// TIA Portal V16 export
// export: Created 2022-11-14T17:35:39.342922Z, ExportSetting WithDefaults, DisplayName Totally Integrated Automation Portal, DisplayVersion V16, DisplayName TIA Portal Version Control Interface, DisplayVersion V16, DisplayName TIA Portal Openness, DisplayVersion V16, DisplayName STEP 7 Professional, DisplayVersion V16, DisplayName STEP 7 Safety, DisplayVersion V16, DisplayName WinCC Advanced, DisplayVersion V16
DATA_BLOCK "Timer"   // DB2
{ S7_Optimized_Access := 'TRUE' }
VERSION : 0.0
// stored: AutoNumber false, IsOnlyStoredInLoadMemory false, IsRetainMemResEnabled false, IsWriteProtectedInAS false, MemoryReserve 100
   VAR
      T0 { S7_SetPoint := 'True'} : IEC_TIMER;   // Delay on pallet positioning
      T1 { S7_SetPoint := 'True'} : IEC_TIMER;   // Timer for acoustic siren
      T2 { S7_SetPoint := 'True'} : IEC_TIMER;   // Timer for restart after emergency
      T3 { S7_SetPoint := 'True'} : IEC_TIMER;   // Timer to reset emergency
      T4 { S7_SetPoint := 'True'} : IEC_TIMER;   // Timer to reset the cycles
      T5 { S7_SetPoint := 'True'} : IEC_TIMER;   // Delay for backward on table rotation inverter
      T6 { S7_SetPoint := 'True'} : IEC_TIMER;   // Delay for forward on table rotation inverter
      T7 { S7_SetPoint := 'True'} : IEC_TIMER;   // Timeout for table phase
      T8 { S7_SetPoint := 'True'} : IEC_TIMER;   // Table rotation speed timer
      T9 { S7_SetPoint := 'True'} : IEC_TIMER;   // Timer SA type for spool carriage motor
      T10 { S7_SetPoint := 'True'} : IEC_TIMER;   // Timer SA type for table rotation motor
      T11 { S7_SetPoint := 'True'} : IEC_TIMER;   // Timer SA type for spool carriage downward
      T12 { S7_SetPoint := 'True'} : IEC_TIMER;   // Timer SA type for spool carriage upward
      T13 { S7_SetPoint := 'True'} : IEC_TIMER;   // Timer SA type for top carriage motor
      T14 { S7_SetPoint := 'True'} : IEC_TIMER;   // Delay for forward on spool carriage and machine conveyor inverter
      T15 { S7_SetPoint := 'True'} : IEC_TIMER;   // Timer for lifter upward
      T16 { S7_SetPoint := 'True'} : IEC_TIMER;   // Timeout for pallet lifter upward/downward
      T17 { S7_SetPoint := 'True'} : IEC_TIMER;   // Time for pressure plate downward
      T18 { S7_SetPoint := 'True'} : IEC_TIMER;   // Timeout for pressure plate upward/downward
      T19 { S7_SetPoint := 'True'} : IEC_TIMER;   // Delay for backward on spool carriage and machine conveyor inverter
      T20 { S7_SetPoint := 'True'} : IEC_TIMER;   // Delay for table rotation deceleration
      T21 { S7_SetPoint := 'True'} : IEC_TIMER;   // Film broken delay for spool carriage
      T22 { S7_SetPoint := 'True'} : IEC_TIMER;   // Delay for pressure plate positioning on pallet
      T23 { S7_SetPoint := 'True'} : IEC_TIMER;   // Timer SA type for conveyor motor
      T24 { S7_SetPoint := 'True'} : IEC_TIMER;   // Delay on pallet positioning left
      T25 { S7_SetPoint := 'True'} : IEC_TIMER;   // Delay on machine conveyor stop
      T26 { S7_SetPoint := 'True'} : IEC_TIMER;   // Delay to load/unload pallet simultaneously
      T27 { S7_SetPoint := 'True'} : IEC_TIMER;   // Delay to have outfeed control free
      T28 { S7_SetPoint := 'True'} : IEC_TIMER;   // Timer for end of transfer signal
      T29 { S7_SetPoint := 'True'} : IEC_TIMER;   // Timer to check spool carriage encoder
      T30 { S7_SetPoint := 'True'} : IEC_TIMER;   // Timer to check spool carriage encoder
      T31 { S7_SetPoint := 'True'} : IEC_TIMER;   // Time to record spool carriage movement speed
      T32 { S7_SetPoint := 'True'} : IEC_TIMER;   // Timeout for single or lower(double) rope unit open/close
      T33 { S7_SetPoint := 'True'} : IEC_TIMER;   // Timer for outfeed rotating table control engaged
      T34 { S7_SetPoint := 'True'} : IEC_TIMER;   // Timer for prestretch restart
      T35 { S7_SetPoint := 'True'} : IEC_TIMER;   // Delay to open single or lower(double) rope unit
      T36 { S7_SetPoint := 'True'} : IEC_TIMER;   // Timeout for welder unit upward/downward
      T37 { S7_SetPoint := 'True'} : IEC_TIMER;   // Timeout for welder contrast downward
      T38 { S7_SetPoint := 'True'} : IEC_TIMER;   // Timeout for welder contrast upward
      T39 { S7_SetPoint := 'True'} : IEC_TIMER;   // Timeout for clamp upward/downward
      T40 { S7_SetPoint := 'True'} : IEC_TIMER;   // Timeout for clamp open/close
      T41 { S7_SetPoint := 'True'} : IEC_TIMER;   // Welding timer for welder
      T42 { S7_SetPoint := 'True'} : IEC_TIMER;   // Cutting timer
      T43 { S7_SetPoint := 'True'} : IEC_TIMER;   // Welder cooler timer
      T44 { S7_SetPoint := 'True'} : IEC_TIMER;   // Timer to check welder circuit 1 (current on)
      T45 { S7_SetPoint := 'True'} : IEC_TIMER;   // Timer to check welder circuit 2 (current off)
      T46 { S7_SetPoint := 'True'} : IEC_TIMER;   // Spring clamp up
      T47 { S7_SetPoint := 'True'} : IEC_TIMER;   // Welder contrast up
      T48 { S7_SetPoint := 'True'} : IEC_TIMER;   // Spring clamp open
      T49 { S7_SetPoint := 'True'} : IEC_TIMER;   // Welder and cut unit up
      T50 { S7_SetPoint := 'True'} : IEC_TIMER;   // Timer for encoder check
      T51 { S7_SetPoint := 'True'} : IEC_TIMER;   // Timer for display comunication control
      T52 { S7_SetPoint := 'True'} : IEC_TIMER;   // Timer to return to page 1 after 3 minutes
      T53 { S7_SetPoint := 'True'} : IEC_TIMER;   // Delay for test cycle
      T54 { S7_SetPoint := 'True'} : IEC_TIMER;   // Timer to reset infeed safety barrier
      T55 { S7_SetPoint := 'True'} : IEC_TIMER;   // Timer to reset infeed safety barrier
      T56 { S7_SetPoint := 'True'} : IEC_TIMER;   // Timer to reset outfeed safety barrier
      T57 { S7_SetPoint := 'True'} : IEC_TIMER;   // Timer to reset outfeed safety barrier
      T58 { S7_SetPoint := 'True'} : IEC_TIMER;   // Delay for infeed safety barrier muting photocell
      T59 { S7_SetPoint := 'True'} : IEC_TIMER;   // Delay for outfeed safety barrier muting photocell
      T60 { S7_SetPoint := 'True'} : IEC_TIMER;   // Delay for spool carriage downward for film tail
      T61 { S7_SetPoint := 'True'} : IEC_TIMER;   // Delay to open clamp during wrapping cycle
      T62 { S7_SetPoint := 'True'} : IEC_TIMER;   // Timer for table rotation forward on twist
      T63 { S7_SetPoint := 'True'} : IEC_TIMER;   // Timer SA type for top carriage upward
      T64 { S7_SetPoint := 'True'} : IEC_TIMER;   // Timer SA type for top carriage downward
      T65 { S7_SetPoint := 'True'} : IEC_TIMER;   // Delay on safety for top carriage movement
      T66 { S7_SetPoint := 'True'} : IEC_TIMER;   // Timer to check top film presence
      T67 { S7_SetPoint := 'True'} : IEC_TIMER;   // Timer to check top film presence
      T68 { S7_SetPoint := 'True'} : IEC_TIMER;   // Timeout for top film cutter forward/backward
      T69 { S7_SetPoint := 'True'} : IEC_TIMER;   // Timeout for clamp to lift top film open/close
      T70 { S7_SetPoint := 'True'} : IEC_TIMER;   // Timeout for clamp to block top film open/close
      T71 { S7_SetPoint := 'True'} : IEC_TIMER;   // Timeout for top carriage forward/backward movement
      T72 { S7_SetPoint := 'True'} : IEC_TIMER;   // Timeout for top carriage forward/backward movement
      T73 { S7_SetPoint := 'True'} : IEC_TIMER;   // Timeout for top carriage upward/downward movement
      T74 { S7_SetPoint := 'True'} : IEC_TIMER;   // Timeout for top carriage upward/downward movement
      T75 { S7_SetPoint := 'True'} : IEC_TIMER;   // Delay for spool carriage downward during top cycle
      T76 { S7_SetPoint := 'True'} : IEC_TIMER;   // Claw clamp closed
      T77 { S7_SetPoint := 'True'} : IEC_TIMER;   // Timeout for welder and cut unit forward/backward
      T78 { S7_SetPoint := 'True'} : IEC_TIMER;   // Delay to open upper(double) rope unit
      T79 { S7_SetPoint := 'True'} : IEC_TIMER;   // Timer SA type for table rotation brake
      T80 { S7_SetPoint := 'True'} : IEC_TIMER;   // Timer for spool carriage movement speed
      T81 { S7_SetPoint := 'True'} : IEC_TIMER;   // Claw clamp closed
      T82 { S7_SetPoint := 'True'} : IEC_TIMER;   // Timeout for welder and cut unit forward/backward
      T83 { S7_SetPoint := 'True'} : IEC_TIMER;   // Delay between airblow and clamp
      T84 { S7_SetPoint := 'True'} : IEC_TIMER;   // Timer for table rotation speed
      T85 { S7_SetPoint := 'True'} : IEC_TIMER;   // Delay on infeed conveyor stop
      T86 { S7_SetPoint := 'True'} : IEC_TIMER;   // Delay for prestretch during acceleration
      T87 { S7_SetPoint := 'True'} : IEC_TIMER;   // Timer for slow conveyor manual movement
      T88 { S7_SetPoint := 'True'} : IEC_TIMER;
      T89 { S7_SetPoint := 'True'} : IEC_TIMER;   // Timer for wrong pallet positioning without outfeed control
      T90 { S7_SetPoint := 'True'} : IEC_TIMER;   // Timer for spool carriage upward for table cycle
      T91 { S7_SetPoint := 'True'} : IEC_TIMER;   // Delay to close clamp after cutter forward
      T92 { S7_SetPoint := 'True'} : IEC_TIMER;   // Delay for contrast downward
      T93 { S7_SetPoint := 'True'} : IEC_TIMER;
      T94 { S7_SetPoint := 'True'} : IEC_TIMER;
      T95 { S7_SetPoint := 'True'} : IEC_TIMER;
      T96 { S7_SetPoint := 'True'} : IEC_TIMER;   // Timeout for fire door pos.4-5 opening
      T97 { S7_SetPoint := 'True'} : IEC_TIMER;   // Delay conveyor manual movement
      T98 { S7_SetPoint := 'True'} : IEC_TIMER;   // Delay start cycle pos.1
      T99 { S7_SetPoint := 'True'} : IEC_TIMER;   // Time to load with forklift
      T100 { S7_SetPoint := 'True'} : IEC_TIMER;   // Timer for end of pallet transfer in infeed signal
      T101 { S7_SetPoint := 'True'} : IEC_TIMER;   // Timeout for conveyor pos 01
      T102 { S7_SetPoint := 'True'} : IEC_TIMER;   // Time to load with forklift
      T103 { S7_SetPoint := 'True'} : IEC_TIMER;   // Timeout for conveyor pos 02
      T104 { S7_SetPoint := 'True'} : IEC_TIMER;
      T105 { S7_SetPoint := 'True'} : IEC_TIMER;   // Timeout for conveyor pos 04
      T106 { S7_SetPoint := 'True'} : IEC_TIMER;   // Timeout for conveyor pos 03
      T107 { S7_SetPoint := 'True'} : IEC_TIMER;   // Time for pallet unload with forklift
      T108 { S7_SetPoint := 'True'} : IEC_TIMER;   // Delay Button Stop cycle support memory
      T109 { S7_SetPoint := 'True'} : IEC_TIMER;   // Time for pallet load with forklift from reverse
      T110 { S7_SetPoint := 'True'} : IEC_TIMER;   // Timer to reset machine and cycle
      T111 { S7_SetPoint := 'True'} : IEC_TIMER;   // Delay timer for lifter pos.2 low position
      T112 { S7_SetPoint := 'True'} : IEC_TIMER;   // Delay timer for lifter pos.2 up position
      T113 { S7_SetPoint := 'True'} : IEC_TIMER;   // Delay timer pallet positioned on lifter pos.2
      T114 { S7_SetPoint := 'True'} : IEC_TIMER;   // Timer SA for lifter in top position
      T115 { S7_SetPoint := 'True'} : IEC_TIMER;   // Timeout for conveyor pos.2
      T116 { S7_SetPoint := 'True'} : IEC_TIMER;   // Timeout for lifter pos.2 upstroke
      T117 { S7_SetPoint := 'True'} : IEC_TIMER;   // Timeout for lifter pos.2 downstroke
      T118 { S7_SetPoint := 'True'} : IEC_TIMER;   // Timer to filter lifter pos.2 in up position
      T119 { S7_SetPoint := 'True'} : IEC_TIMER;
      T120 { S7_SetPoint := 'True'} : IEC_TIMER;   // Timer to check conveyor encoder
      T121 { S7_SetPoint := 'True'} : IEC_TIMER;   // Timer to check conveyor encoder
      T122 { S7_SetPoint := 'True'} : IEC_TIMER;
      T123 { S7_SetPoint := 'True'} : IEC_TIMER;
      T124 { S7_SetPoint := 'True'} : IEC_TIMER;
      T125 { S7_SetPoint := 'True'} : IEC_TIMER;
      T126 { S7_SetPoint := 'True'} : IEC_TIMER;
      T127 { S7_SetPoint := 'True'} : IEC_TIMER;   // Delay to have outfeed rotating arm control free from reverse
      T128 { S7_SetPoint := 'True'} : IEC_TIMER;   // Timer for end of transfer signal from reverse
      T129 { S7_SetPoint := 'True'} : IEC_TIMER;
      T130 { S7_SetPoint := 'True'} : IEC_TIMER;
      T131 { S7_SetPoint := 'True'} : IEC_TIMER;
      T132 { S7_SetPoint := 'True'} : IEC_TIMER;   // Timeout for single or lower(double) rope unit open/close
      T133 { S7_SetPoint := 'True'} : IEC_TIMER;
      T134 { S7_SetPoint := 'True'} : IEC_TIMER;
      T135 { S7_SetPoint := 'True'} : IEC_TIMER;   // Delay to open single or lower(double) rope unit
      T136 { S7_SetPoint := 'True'} : IEC_TIMER;
      T137 { S7_SetPoint := 'True'} : IEC_TIMER;
      T138 { S7_SetPoint := 'True'} : IEC_TIMER;
      T139 { S7_SetPoint := 'True'} : IEC_TIMER;   // Delay for top carriage forward stop (Top)
      T140 { S7_SetPoint := 'True'} : IEC_TIMER;   // Delay for top carriage backward stop (Top)
      T141 { S7_SetPoint := 'True'} : IEC_TIMER;
      T142 { S7_SetPoint := 'True'} : IEC_TIMER;   // Delay for top carriage down to release top film (Top)
      T143 { S7_SetPoint := 'True'} : IEC_TIMER;   // Delay to release top film from clamp (Top)
      T144 { S7_SetPoint := 'True'} : IEC_TIMER;   // Timer 1 for top film broken (Top)
      T145 { S7_SetPoint := 'True'} : IEC_TIMER;   // Timer 2 for top film broken (Top)
      T146 { S7_SetPoint := 'True'} : IEC_TIMER;   // Delay to stop top carriage forward for top film broken (Top)
      T147 { S7_SetPoint := 'True'} : IEC_TIMER;   // Delay to stop top carriage against vibration (Top)
      T148 { S7_SetPoint := 'True'} : IEC_TIMER;   // Timeout for top cutter (Top)
      T149 { S7_SetPoint := 'True'} : IEC_TIMER;   // Timeout for clamp to pull top film (Top)
      T150 { S7_SetPoint := 'True'} : IEC_TIMER;   // Timeout for clamp to block top film (Top)
      T151 { S7_SetPoint := 'True'} : IEC_TIMER;   // Timer SA type for top brake (Top)
      T152 { S7_SetPoint := 'True'} : IEC_TIMER;   // Timer for top brake control (Top)
      T153 { S7_SetPoint := 'True'} : IEC_TIMER;
      T154 { S7_SetPoint := 'True'} : IEC_TIMER;
      T155 { S7_SetPoint := 'True'} : IEC_TIMER;   // Timeout for conveyor pos 03
      T156 { S7_SetPoint := 'True'} : IEC_TIMER;   // Timeout for conveyor pos 04
      T157 { S7_SetPoint := 'True'} : IEC_TIMER;   // Timeout for conveyor pos 05
      T158 { S7_SetPoint := 'True'} : IEC_TIMER;   // Timeout for conveyor pos 06
      T159 { S7_SetPoint := 'True'} : IEC_TIMER;   // Timeout for conveyor pos 07
      T160 { S7_SetPoint := 'True'} : IEC_TIMER;   // Timeout for conveyor pos 08
      T161 { S7_SetPoint := 'True'} : IEC_TIMER;
      T162 { S7_SetPoint := 'True'} : IEC_TIMER;
      T163 { S7_SetPoint := 'True'} : IEC_TIMER;   // Watchdog timer for network communication
      T164 { S7_SetPoint := 'True'} : IEC_TIMER;
      T165 { S7_SetPoint := 'True'} : IEC_TIMER;
      T166 { S7_SetPoint := 'True'} : IEC_TIMER;
      T167 { S7_SetPoint := 'True'} : IEC_TIMER;
      T168 { S7_SetPoint := 'True'} : IEC_TIMER;
      T169 { S7_SetPoint := 'True'} : IEC_TIMER;
      T170 { S7_SetPoint := 'True'} : IEC_TIMER;
      T171 { S7_SetPoint := 'True'} : IEC_TIMER;
      T172 { S7_SetPoint := 'True'} : IEC_TIMER;
      T173 { S7_SetPoint := 'True'} : IEC_TIMER;
      T174 { S7_SetPoint := 'True'} : IEC_TIMER;
      T175 { S7_SetPoint := 'True'} : IEC_TIMER;
      T176 { S7_SetPoint := 'True'} : IEC_TIMER;
      T177 { S7_SetPoint := 'True'} : IEC_TIMER;
      T178 { S7_SetPoint := 'True'} : IEC_TIMER;
      T179 { S7_SetPoint := 'True'} : IEC_TIMER;   // Delay for top pallet height reading photocell (fast cycle)
      T180 { S7_SetPoint := 'True'} : IEC_TIMER;
      T181 { S7_SetPoint := 'True'} : IEC_TIMER;
      T182 { S7_SetPoint := 'True'} : IEC_TIMER;
      T183 { S7_SetPoint := 'True'} : IEC_TIMER;
      T184 { S7_SetPoint := 'True'} : IEC_TIMER;
      T185 { S7_SetPoint := 'True'} : IEC_TIMER;
      T186 { S7_SetPoint := 'True'} : IEC_TIMER;
      T187 { S7_SetPoint := 'True'} : IEC_TIMER;
      T188 { S7_SetPoint := 'True'} : IEC_TIMER;
      T189 { S7_SetPoint := 'True'} : IEC_TIMER;
      T190 { S7_SetPoint := 'True'} : IEC_TIMER;
      T191 { S7_SetPoint := 'True'} : IEC_TIMER;
      T192 { S7_SetPoint := 'True'} : IEC_TIMER;
      T193 { S7_SetPoint := 'True'} : IEC_TIMER;
      T194 { S7_SetPoint := 'True'} : IEC_TIMER;
      T195 { S7_SetPoint := 'True'} : IEC_TIMER;
      T196 { S7_SetPoint := 'True'} : IEC_TIMER;
      T197 { S7_SetPoint := 'True'} : IEC_TIMER;
      T198 { S7_SetPoint := 'True'} : IEC_TIMER;
      T199 { S7_SetPoint := 'True'} : IEC_TIMER;
      T200 { S7_SetPoint := 'True'} : IEC_TIMER;   // T_InverterAlarm - Time to filter inverter alarms
      T201 { S7_SetPoint := 'True'} : IEC_TIMER;   // T_ProfinetDiag - Time to filter 'DeviceStates' diagnostic output (Profinet)
      T202 { S7_SetPoint := 'True'} : IEC_TIMER;   // Timer for U201 start command (after enable)
      T203 { S7_SetPoint := 'True'} : IEC_TIMER;   // Timer table backward
      T204 { S7_SetPoint := 'True'} : IEC_TIMER;   // Timer ciclo fiera
      T205 { S7_SetPoint := 'True'} : IEC_TIMER;   // TON per OFF1 U201
      T206 { S7_SetPoint := 'True'} : IEC_TIMER;   // TOF per OFF1 U201
      T207 { S7_SetPoint := 'True'} : IEC_TIMER;   // Timer coppia tavola
      T208 { S7_SetPoint := 'True'} : IEC_TIMER;   // T_ModbusErrors
      T209 { S7_SetPoint := 'True'} : IEC_TIMER;
      T210 { S7_SetPoint := 'True'} : IEC_TIMER;   // Time to filter contrast back sensor
      T211 { S7_SetPoint := 'True'} : IEC_TIMER;   // Timeout for welder contrast forward
      T212 { S7_SetPoint := 'True'} : IEC_TIMER;   // Timeout for welder contrast backward
      T213 { S7_SetPoint := 'True'} : IEC_TIMER;   // Timeout for (double) full rope unit open/close
      T214 { S7_SetPoint := 'True'} : IEC_TIMER;   // Delay to open single or lower(double) rope unit
      T215 { S7_SetPoint := 'True'} : IEC_TIMER;   // Time Contrast Backward
      T216 { S7_SetPoint := 'True'} : IEC_TIMER;   // Time Contrast Manual forward
   END_VAR
BEGIN
   T0.PT := T#0MS;
   T0.IN := FALSE;
   T1.PT := T#1S_200MS;
   T1.IN := FALSE;
   T2.PT := T#6S;
   T2.IN := TRUE;
   T3.PT := T#700MS;
   T3.IN := FALSE;
   T4.PT := T#2S;
   T4.IN := FALSE;
   T5.PT := T#800MS;
   T5.IN := FALSE;
   T6.PT := T#800MS;
   T6.IN := FALSE;
   T7.PT := T#50S;
   T7.IN := FALSE;
   T8.PT := T#1M_39S;
   T8.IN := FALSE;
   T9.PT := T#700MS;
   T9.IN := FALSE;
   T10.PT := T#2S;
   T10.IN := FALSE;
   T11.PT := T#500MS;
   T11.IN := FALSE;
   T12.PT := T#500MS;
   T12.IN := FALSE;
   T13.PT := T#0MS;
   T13.IN := FALSE;
   T14.PT := T#200MS;
   T14.IN := FALSE;
   T15.PT := T#0MS;
   T15.IN := FALSE;
   T16.PT := T#0MS;
   T16.IN := FALSE;
   T17.PT := T#0MS;
   T17.IN := FALSE;
   T18.PT := T#0MS;
   T18.IN := FALSE;
   T19.PT := T#200MS;
   T19.IN := FALSE;
   T20.PT := T#0MS;
   T20.IN := FALSE;
   T21.PT := T#2S;
   T21.IN := FALSE;
   T22.PT := T#0MS;
   T22.IN := FALSE;
   T23.PT := T#0MS;
   T23.IN := FALSE;
   T24.PT := T#0MS;
   T24.IN := FALSE;
   T25.PT := T#0MS;
   T25.IN := FALSE;
   T26.PT := T#0MS;
   T26.IN := FALSE;
   T27.PT := T#1S_500MS;
   T27.IN := TRUE;
   T28.PT := T#2S;
   T28.IN := TRUE;
   T29.PT := T#0MS;
   T29.IN := FALSE;
   T30.PT := T#3S;
   T30.IN := FALSE;
   T31.PT := T#0MS;
   T31.IN := FALSE;
   T32.PT := T#0MS;
   T32.IN := FALSE;
   T33.PT := T#0MS;
   T33.IN := FALSE;
   T34.PT := T#0MS;
   T34.IN := FALSE;
   T35.PT := T#0MS;
   T35.IN := FALSE;
   T36.PT := T#0MS;
   T36.IN := FALSE;
   T37.PT := T#0MS;
   T37.IN := FALSE;
   T38.PT := T#10S;
   T38.IN := FALSE;
   T39.PT := T#0MS;
   T39.IN := FALSE;
   T40.PT := T#0MS;
   T40.IN := FALSE;
   T41.PT := T#650MS;
   T41.IN := FALSE;
   T42.PT := T#3S;
   T42.IN := FALSE;
   T43.PT := T#0MS;
   T43.IN := FALSE;
   T44.PT := T#3S_500MS;
   T44.IN := FALSE;
   T45.PT := T#1S;
   T45.IN := FALSE;
   T46.PT := T#0MS;
   T46.IN := FALSE;
   T47.PT := T#500MS;
   T47.IN := TRUE;
   T48.PT := T#0MS;
   T48.IN := FALSE;
   T49.PT := T#0MS;
   T49.IN := FALSE;
   T50.PT := T#0MS;
   T50.IN := FALSE;
   T51.PT := T#4S;
   T51.IN := TRUE;
   T52.PT := T#0MS;
   T52.IN := FALSE;
   T53.PT := T#0MS;
   T53.IN := TRUE;
   T54.PT := T#0MS;
   T54.IN := FALSE;
   T55.PT := T#0MS;
   T55.IN := FALSE;
   T56.PT := T#0MS;
   T56.IN := FALSE;
   T57.PT := T#0MS;
   T57.IN := FALSE;
   T58.PT := T#0MS;
   T58.IN := FALSE;
   T59.PT := T#0MS;
   T59.IN := FALSE;
   T60.PT := T#0MS;
   T60.IN := FALSE;
   T61.PT := T#0MS;
   T61.IN := FALSE;
   T62.PT := T#0MS;
   T62.IN := FALSE;
   T63.PT := T#0MS;
   T63.IN := FALSE;
   T64.PT := T#0MS;
   T64.IN := FALSE;
   T65.PT := T#0MS;
   T65.IN := FALSE;
   T66.PT := T#0MS;
   T66.IN := FALSE;
   T67.PT := T#0MS;
   T67.IN := FALSE;
   T68.PT := T#0MS;
   T68.IN := FALSE;
   T69.PT := T#0MS;
   T69.IN := FALSE;
   T70.PT := T#0MS;
   T70.IN := FALSE;
   T71.PT := T#0MS;
   T71.IN := FALSE;
   T72.PT := T#0MS;
   T72.IN := FALSE;
   T73.PT := T#0MS;
   T73.IN := FALSE;
   T74.PT := T#0MS;
   T74.IN := FALSE;
   T75.PT := T#0MS;
   T75.IN := FALSE;
   T76.PT := T#0MS;
   T76.IN := FALSE;
   T77.PT := T#0MS;
   T77.IN := FALSE;
   T78.PT := T#0MS;
   T78.IN := FALSE;
   T79.PT := T#2S;
   T79.IN := FALSE;
   T80.PT := T#1S;
   T80.IN := TRUE;
   T81.PT := T#700MS;
   T81.IN := TRUE;
   T82.PT := T#10S;
   T82.IN := FALSE;
   T83.PT := T#500MS;
   T83.IN := FALSE;
   T84.PT := T#400MS;
   T84.IN := TRUE;
   T85.PT := T#0MS;
   T85.IN := FALSE;
   T86.PT := T#300MS;
   T86.IN := FALSE;
   T87.PT := T#0MS;
   T87.IN := FALSE;
   T88.PT := T#0MS;
   T88.IN := FALSE;
   T89.PT := T#0MS;
   T89.IN := FALSE;
   T90.PT := T#2S;
   T90.IN := FALSE;
   T91.PT := T#1S;
   T91.IN := FALSE;
   T92.PT := T#0MS;
   T92.IN := FALSE;
   T93.PT := T#0MS;
   T93.IN := FALSE;
   T94.PT := T#0MS;
   T94.IN := FALSE;
   T95.PT := T#0MS;
   T95.IN := FALSE;
   T96.PT := T#0MS;
   T96.IN := FALSE;
   T97.PT := T#0MS;
   T97.IN := FALSE;
   T98.PT := T#0MS;
   T98.IN := FALSE;
   T99.PT := T#0MS;
   T99.IN := FALSE;
   T100.PT := T#0MS;
   T100.IN := FALSE;
   T101.PT := T#0MS;
   T101.IN := FALSE;
   T102.PT := T#0MS;
   T102.IN := FALSE;
   T103.PT := T#0MS;
   T103.IN := FALSE;
   T104.PT := T#0MS;
   T104.IN := FALSE;
   T105.PT := T#0MS;
   T105.IN := FALSE;
   T106.PT := T#0MS;
   T106.IN := FALSE;
   T107.PT := T#0MS;
   T107.IN := FALSE;
   T108.PT := T#0MS;
   T108.IN := FALSE;
   T109.PT := T#0MS;
   T109.IN := FALSE;
   T110.PT := T#0MS;
   T110.IN := FALSE;
   T111.PT := T#0MS;
   T111.IN := FALSE;
   T112.PT := T#0MS;
   T112.IN := FALSE;
   T113.PT := T#0MS;
   T113.IN := FALSE;
   T114.PT := T#0MS;
   T114.IN := FALSE;
   T115.PT := T#0MS;
   T115.IN := FALSE;
   T116.PT := T#0MS;
   T116.IN := FALSE;
   T117.PT := T#0MS;
   T117.IN := FALSE;
   T118.PT := T#0MS;
   T118.IN := FALSE;
   T119.PT := T#0MS;
   T119.IN := FALSE;
   T120.PT := T#0MS;
   T120.IN := FALSE;
   T121.PT := T#0MS;
   T121.IN := FALSE;
   T122.PT := T#0MS;
   T122.IN := FALSE;
   T123.PT := T#0MS;
   T123.IN := FALSE;
   T124.PT := T#0MS;
   T124.IN := FALSE;
   T125.PT := T#0MS;
   T125.IN := FALSE;
   T126.PT := T#0MS;
   T126.IN := FALSE;
   T127.PT := T#0MS;
   T127.IN := FALSE;
   T128.PT := T#0MS;
   T128.IN := FALSE;
   T129.PT := T#0MS;
   T129.IN := FALSE;
   T130.PT := T#0MS;
   T130.IN := FALSE;
   T131.PT := T#0MS;
   T131.IN := FALSE;
   T132.PT := T#3S;
   T132.IN := FALSE;
   T133.PT := T#0MS;
   T133.IN := FALSE;
   T134.PT := T#0MS;
   T134.IN := FALSE;
   T135.PT := T#1S_500MS;
   T135.IN := TRUE;
   T136.PT := T#0MS;
   T136.IN := FALSE;
   T137.PT := T#0MS;
   T137.IN := FALSE;
   T138.PT := T#0MS;
   T138.IN := FALSE;
   T139.PT := T#0MS;
   T139.IN := FALSE;
   T140.PT := T#0MS;
   T140.IN := FALSE;
   T141.PT := T#0MS;
   T141.IN := FALSE;
   T142.PT := T#0MS;
   T142.IN := FALSE;
   T143.PT := T#0MS;
   T143.IN := FALSE;
   T144.PT := T#0MS;
   T144.IN := FALSE;
   T145.PT := T#0MS;
   T145.IN := FALSE;
   T146.PT := T#0MS;
   T146.IN := FALSE;
   T147.PT := T#0MS;
   T147.IN := FALSE;
   T148.PT := T#0MS;
   T148.IN := FALSE;
   T149.PT := T#0MS;
   T149.IN := FALSE;
   T150.PT := T#0MS;
   T150.IN := FALSE;
   T151.PT := T#0MS;
   T151.IN := FALSE;
   T152.PT := T#0MS;
   T152.IN := FALSE;
   T153.PT := T#0MS;
   T153.IN := FALSE;
   T154.PT := T#0MS;
   T154.IN := FALSE;
   T155.PT := T#0MS;
   T155.IN := FALSE;
   T156.PT := T#0MS;
   T156.IN := FALSE;
   T157.PT := T#0MS;
   T157.IN := FALSE;
   T158.PT := T#0MS;
   T158.IN := FALSE;
   T159.PT := T#0MS;
   T159.IN := FALSE;
   T160.PT := T#0MS;
   T160.IN := FALSE;
   T161.PT := T#0MS;
   T161.IN := FALSE;
   T162.PT := T#0MS;
   T162.IN := FALSE;
   T163.PT := T#0MS;
   T163.IN := FALSE;
   T164.PT := T#0MS;
   T164.IN := FALSE;
   T165.PT := T#0MS;
   T165.IN := FALSE;
   T166.PT := T#0MS;
   T166.IN := FALSE;
   T167.PT := T#0MS;
   T167.IN := FALSE;
   T168.PT := T#0MS;
   T168.IN := FALSE;
   T169.PT := T#0MS;
   T169.IN := FALSE;
   T170.PT := T#0MS;
   T170.IN := FALSE;
   T171.PT := T#0MS;
   T171.IN := FALSE;
   T172.PT := T#0MS;
   T172.IN := FALSE;
   T173.PT := T#0MS;
   T173.IN := FALSE;
   T174.PT := T#0MS;
   T174.IN := FALSE;
   T175.PT := T#0MS;
   T175.IN := FALSE;
   T176.PT := T#0MS;
   T176.IN := FALSE;
   T177.PT := T#0MS;
   T177.IN := FALSE;
   T178.PT := T#0MS;
   T178.IN := FALSE;
   T179.PT := T#0MS;
   T179.IN := FALSE;
   T180.PT := T#0MS;
   T180.IN := FALSE;
   T181.PT := T#0MS;
   T181.IN := FALSE;
   T182.PT := T#0MS;
   T182.IN := FALSE;
   T183.PT := T#0MS;
   T183.IN := FALSE;
   T184.PT := T#0MS;
   T184.IN := FALSE;
   T185.PT := T#0MS;
   T185.IN := FALSE;
   T186.PT := T#0MS;
   T186.IN := FALSE;
   T187.PT := T#0MS;
   T187.IN := FALSE;
   T188.PT := T#0MS;
   T188.IN := FALSE;
   T189.PT := T#0MS;
   T189.IN := FALSE;
   T190.PT := T#0MS;
   T190.IN := FALSE;
   T191.PT := T#0MS;
   T191.IN := FALSE;
   T192.PT := T#0MS;
   T192.IN := FALSE;
   T193.PT := T#0MS;
   T193.IN := FALSE;
   T194.PT := T#0MS;
   T194.IN := FALSE;
   T195.PT := T#0MS;
   T195.IN := FALSE;
   T196.PT := T#0MS;
   T196.IN := FALSE;
   T197.PT := T#0MS;
   T197.IN := FALSE;
   T198.PT := T#0MS;
   T198.IN := FALSE;
   T199.PT := T#0MS;
   T199.IN := FALSE;
   T200.PT := T#5S;
   T200.IN := FALSE;
   T201.PT := T#200MS;
   T201.IN := TRUE;
   T202.PT := T#200MS;
   T202.IN := FALSE;
   T203.PT := T#1S;
   T203.IN := FALSE;
   T204.PT := T#0MS;
   T204.IN := FALSE;
   T205.PT := T#200MS;
   T205.IN := FALSE;
   T206.PT := T#200MS;
   T206.IN := FALSE;
   T207.PT := T#200MS;
   T207.IN := TRUE;
   T208.PT := T#0MS;
   T208.IN := FALSE;
   T209.PT := T#0MS;
   T209.IN := FALSE;
   T210.PT := T#200MS;
   T210.IN := FALSE;
   T211.PT := T#10S;
   T211.IN := FALSE;
   T212.PT := T#0MS;
   T212.IN := FALSE;
   T213.PT := T#3S;
   T213.IN := FALSE;
   T214.PT := T#1S_500MS;
   T214.IN := TRUE;
   T215.PT := T#2S;
   T215.IN := FALSE;
   T216.PT := T#5S;
   T216.IN := FALSE;
END_DATA_BLOCK
